{attribute 'qualified_only'}
{attribute 'strict'}
TYPE E_EtherCATStatusCheck :
(
	MACHINE_STATE_UNINITIALIZED_CR800_ETHERCAT_STATUS_CHECK := 0,
	MACHINE_STATE_UNINITIALIZED_CR800_ETHERCAT_STATUS_CHECK_DONE := 10,
	MACHINE_STATE_UNINITIALIZED_CR800_ETHERCAT_ERROR_RESET := 20,
	MACHINE_STATE_UNINITIALIZED_CR800_ETHERCAT_REQUEST_OP_STATE := 30,
	MACHINE_STATE_UNINITIALIZED_CR800_CHECK_POWER_REGISTER := 40
);
END_TYPE

(* stored: Version 1.1.0.1, ProductVersion 3.1.4024.9
   DUT E_EtherCATStatusCheck: Id {62e52f41-3e22-4894-a269-d46933855234} *)
